// TIA Portal V17 export
// export: Created 2025-03-05T08:00:39.2851451Z, ExportSetting WithDefaults, DisplayName Totally Integrated Automation Portal, DisplayVersion V17 Update 8, DisplayName TIA Portal Openness, DisplayVersion V17 Update 8, DisplayName TIA Portal Version Control Interface, DisplayVersion V17, DisplayName SINAMICS Startdrive Advanced, DisplayVersion V17 SP2, DisplayName SINAMICS Startdrive G110M, G120, G120C, G120D, G120P, G115D, DisplayVersion V17 SP2, DisplayName SINAMICS Startdrive G130, G150, S120, S150, SINAMICS MV, S210, DisplayVersion V17 SP2, DisplayName STEP 7 Professional, DisplayVersion V17 Update 8, DisplayName SINUMERIK ONE STEP 7 Toolbox, DisplayVersion V17 Update 12, DisplayName SINUMERIK 840D sl STEP 7 Toolbox, DisplayVersion V17 Update 12, DisplayName STEP 7 Safety, DisplayVersion V17 Update 6, DisplayName WinCC Advanced, DisplayVersion V17 Update 8
FUNCTION "FC1281_UNIT_02_PART_CHECK_STATION" : Void   // FC1281, LAD
{ S7_Optimized_Access := 'TRUE' }
VERSION : 0.1
// stored: AutoNumber false, IsIECCheckEnabled false, SetENOAutomatically false, UDAEnableTagReadback false
   VAR CONSTANT
      FC_NUMBER : Int := 1281;
   END_VAR
   VAR_TEMP   // added for the SCL form of the ladder/FBD networks
      _w1 : Bool;
      _w2 : Bool;
   END_VAR
BEGIN

REGION Network 1: GENERAL CONDITIONS
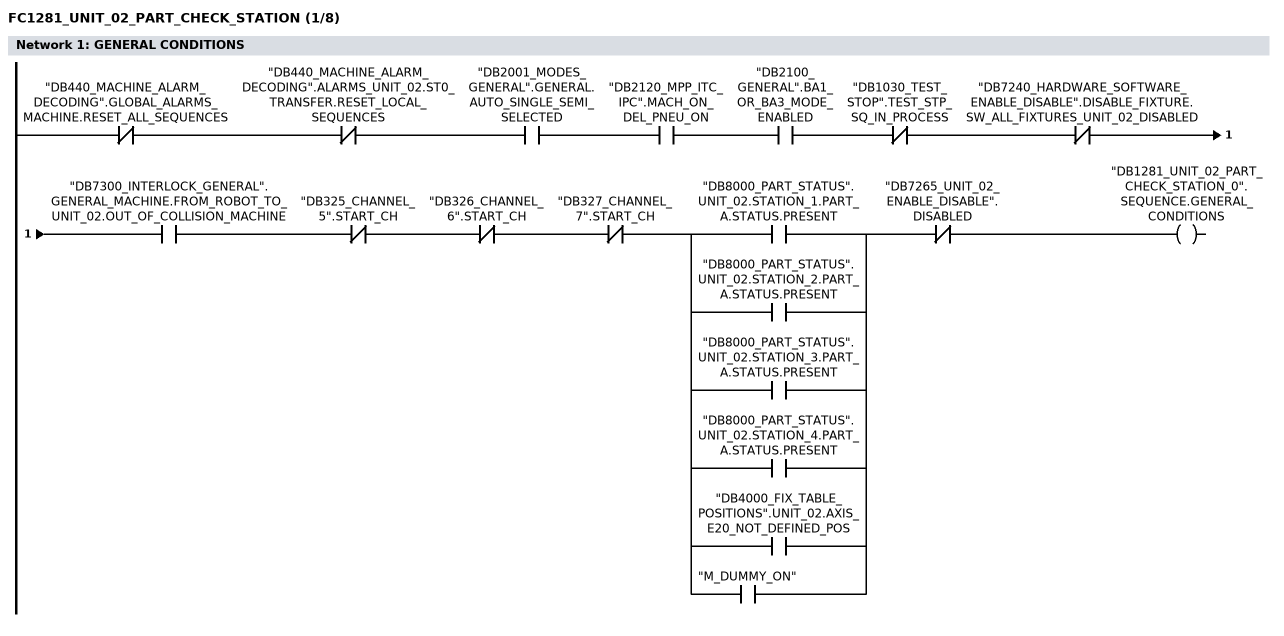
   RUNG wire#powerrail
      I_Contact( "DB440_MACHINE_ALARM_DECODING".GLOBAL_ALARMS_MACHINE.RESET_ALL_SEQUENCES )
      I_Contact( "DB440_MACHINE_ALARM_DECODING".ALARMS_UNIT_02.ST0_TRANSFER.RESET_LOCAL_SEQUENCES )
      Contact( "DB2001_MODES_GENERAL".GENERAL.AUTO_SINGLE_SEMI_SELECTED )
      Contact( "DB2120_MPP_ITC_IPC".MACH_ON_DEL_PNEU_ON )
      Contact( "DB2100_GENERAL".BA1_OR_BA3_MODE_ENABLED )
      I_Contact( "DB1030_TEST_STOP".TEST_STP_SQ_IN_PROCESS )
      I_Contact( "DB7240_HARDWARE_SOFTWARE_ENABLE_DISABLE".DISABLE_FIXTURE.SW_ALL_FIXTURES_UNIT_02_DISABLED )
      Contact( "DB7300_INTERLOCK_GENERAL".GENERAL_MACHINE.FROM_ROBOT_TO_UNIT_02.OUT_OF_COLLISION_MACHINE )
      I_Contact( "DB325_CHANNEL_5".START_CH )
      I_Contact( "DB326_CHANNEL_6".START_CH )
      I_Contact( "DB327_CHANNEL_7".START_CH )
      wire#w1
      Contact( "DB8000_PART_STATUS".UNIT_02.STATION_1.PART_A.STATUS.PRESENT )
      wire#w2
      I_Contact( "DB7265_UNIT_02_ENABLE_DISABLE".DISABLED )
      Coil( "DB1281_UNIT_02_PART_CHECK_STATION_0".SEQUENCE.GENERAL_CONDITIONS )
   END_RUNG
   RUNG wire#w1
      Contact( "DB8000_PART_STATUS".UNIT_02.STATION_2.PART_A.STATUS.PRESENT )
   END_RUNG wire#w2
   RUNG wire#w1
      Contact( "DB8000_PART_STATUS".UNIT_02.STATION_3.PART_A.STATUS.PRESENT )
   END_RUNG wire#w2
   RUNG wire#w1
      Contact( "DB8000_PART_STATUS".UNIT_02.STATION_4.PART_A.STATUS.PRESENT )
   END_RUNG wire#w2
   RUNG wire#w1
      Contact( "DB4000_FIX_TABLE_POSITIONS".UNIT_02.AXIS_E20_NOT_DEFINED_POS )
   END_RUNG wire#w2
   RUNG wire#w1
      Contact( "M_DUMMY_ON" )
   END_RUNG wire#w2
   // the same network as SCL:
   "DB1281_UNIT_02_PART_CHECK_STATION_0".SEQUENCE.GENERAL_CONDITIONS := NOT "DB440_MACHINE_ALARM_DECODING".GLOBAL_ALARMS_MACHINE.RESET_ALL_SEQUENCES AND NOT "DB440_MACHINE_ALARM_DECODING".ALARMS_UNIT_02.ST0_TRANSFER.RESET_LOCAL_SEQUENCES AND "DB2001_MODES_GENERAL".GENERAL.AUTO_SINGLE_SEMI_SELECTED AND "DB2120_MPP_ITC_IPC".MACH_ON_DEL_PNEU_ON AND "DB2100_GENERAL".BA1_OR_BA3_MODE_ENABLED AND NOT "DB1030_TEST_STOP".TEST_STP_SQ_IN_PROCESS AND NOT "DB7240_HARDWARE_SOFTWARE_ENABLE_DISABLE".DISABLE_FIXTURE.SW_ALL_FIXTURES_UNIT_02_DISABLED AND "DB7300_INTERLOCK_GENERAL".GENERAL_MACHINE.FROM_ROBOT_TO_UNIT_02.OUT_OF_COLLISION_MACHINE AND NOT "DB325_CHANNEL_5".START_CH AND NOT "DB326_CHANNEL_6".START_CH AND NOT "DB327_CHANNEL_7".START_CH AND ("DB8000_PART_STATUS".UNIT_02.STATION_1.PART_A.STATUS.PRESENT OR "DB8000_PART_STATUS".UNIT_02.STATION_2.PART_A.STATUS.PRESENT OR "DB8000_PART_STATUS".UNIT_02.STATION_3.PART_A.STATUS.PRESENT OR "DB8000_PART_STATUS".UNIT_02.STATION_4.PART_A.STATUS.PRESENT OR "DB4000_FIX_TABLE_POSITIONS".UNIT_02.AXIS_E20_NOT_DEFINED_POS OR "M_DUMMY_ON") AND NOT "DB7265_UNIT_02_ENABLE_DISABLE".DISABLED;
END_REGION

REGION Network 2: OPERATOR HELP
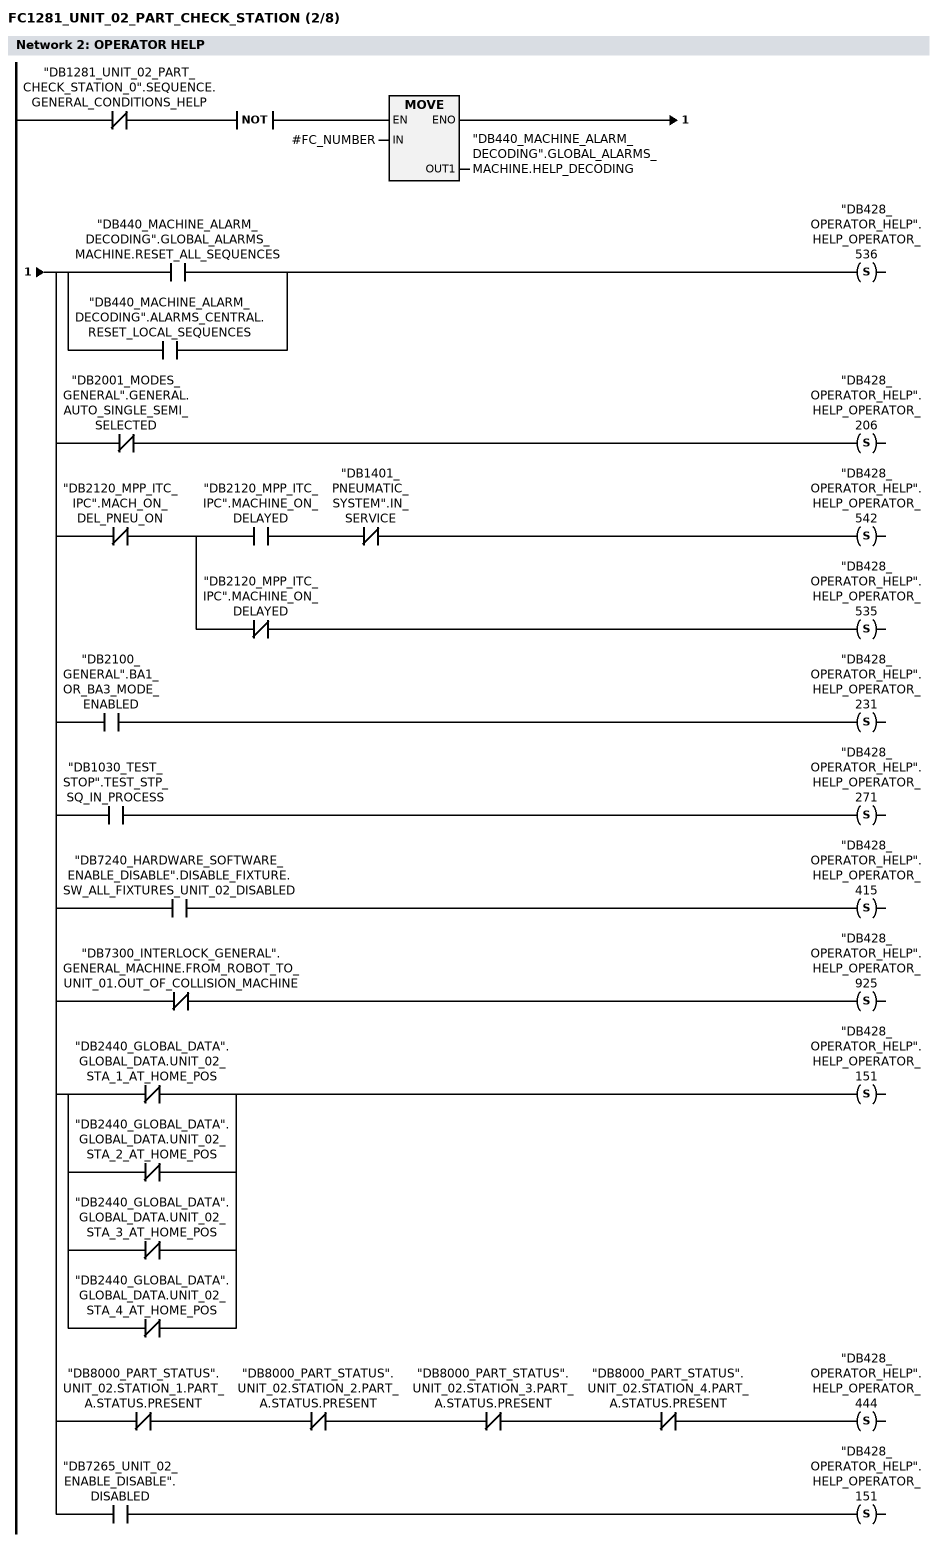
   RUNG wire#powerrail
      I_Contact( "DB1281_UNIT_02_PART_CHECK_STATION_0".SEQUENCE.GENERAL_CONDITIONS_HELP )
      Not()
      { S7_GenerateENO := "TRUE" } Move(in := #FC_NUMBER, out1 => "DB440_MACHINE_ALARM_DECODING".GLOBAL_ALARMS_MACHINE.HELP_DECODING)
      wire#w1
      Contact( "DB440_MACHINE_ALARM_DECODING".GLOBAL_ALARMS_MACHINE.RESET_ALL_SEQUENCES )
      wire#w2
      S_Coil( "DB428_OPERATOR_HELP".HELP_OPERATOR_536 )
   END_RUNG
   RUNG wire#w1
      Contact( "DB440_MACHINE_ALARM_DECODING".ALARMS_CENTRAL.RESET_LOCAL_SEQUENCES )
   END_RUNG wire#w2
   RUNG wire#w1
      I_Contact( "DB2001_MODES_GENERAL".GENERAL.AUTO_SINGLE_SEMI_SELECTED )
      S_Coil( "DB428_OPERATOR_HELP".HELP_OPERATOR_206 )
   END_RUNG
   RUNG wire#w1
      I_Contact( "DB2120_MPP_ITC_IPC".MACH_ON_DEL_PNEU_ON )
      wire#w3
      Contact( "DB2120_MPP_ITC_IPC".MACHINE_ON_DELAYED )
      I_Contact( "DB1401_PNEUMATIC_SYSTEM".IN_SERVICE )
      S_Coil( "DB428_OPERATOR_HELP".HELP_OPERATOR_542 )
   END_RUNG
   RUNG wire#w3
      I_Contact( "DB2120_MPP_ITC_IPC".MACHINE_ON_DELAYED )
      S_Coil( "DB428_OPERATOR_HELP".HELP_OPERATOR_535 )
   END_RUNG
   RUNG wire#w1
      Contact( "DB2100_GENERAL".BA1_OR_BA3_MODE_ENABLED )
      S_Coil( "DB428_OPERATOR_HELP".HELP_OPERATOR_231 )
   END_RUNG
   RUNG wire#w1
      Contact( "DB1030_TEST_STOP".TEST_STP_SQ_IN_PROCESS )
      S_Coil( "DB428_OPERATOR_HELP".HELP_OPERATOR_271 )
   END_RUNG
   RUNG wire#w1
      Contact( "DB7240_HARDWARE_SOFTWARE_ENABLE_DISABLE".DISABLE_FIXTURE.SW_ALL_FIXTURES_UNIT_02_DISABLED )
      S_Coil( "DB428_OPERATOR_HELP".HELP_OPERATOR_415 )
   END_RUNG
   RUNG wire#w1
      I_Contact( "DB7300_INTERLOCK_GENERAL".GENERAL_MACHINE.FROM_ROBOT_TO_UNIT_01.OUT_OF_COLLISION_MACHINE )
      S_Coil( "DB428_OPERATOR_HELP".HELP_OPERATOR_925 )
   END_RUNG
   RUNG wire#w1
      I_Contact( "DB2440_GLOBAL_DATA".GLOBAL_DATA.UNIT_02_STA_1_AT_HOME_POS )
      wire#w4
      S_Coil( "DB428_OPERATOR_HELP".HELP_OPERATOR_151 )
   END_RUNG
   RUNG wire#w1
      I_Contact( "DB2440_GLOBAL_DATA".GLOBAL_DATA.UNIT_02_STA_2_AT_HOME_POS )
   END_RUNG wire#w4
   RUNG wire#w1
      I_Contact( "DB2440_GLOBAL_DATA".GLOBAL_DATA.UNIT_02_STA_3_AT_HOME_POS )
   END_RUNG wire#w4
   RUNG wire#w1
      I_Contact( "DB2440_GLOBAL_DATA".GLOBAL_DATA.UNIT_02_STA_4_AT_HOME_POS )
   END_RUNG wire#w4
   RUNG wire#w1
      I_Contact( "DB8000_PART_STATUS".UNIT_02.STATION_1.PART_A.STATUS.PRESENT )
      I_Contact( "DB8000_PART_STATUS".UNIT_02.STATION_2.PART_A.STATUS.PRESENT )
      I_Contact( "DB8000_PART_STATUS".UNIT_02.STATION_3.PART_A.STATUS.PRESENT )
      I_Contact( "DB8000_PART_STATUS".UNIT_02.STATION_4.PART_A.STATUS.PRESENT )
      S_Coil( "DB428_OPERATOR_HELP".HELP_OPERATOR_444 )
   END_RUNG
   RUNG wire#w1
      Contact( "DB7265_UNIT_02_ENABLE_DISABLE".DISABLED )
      S_Coil( "DB428_OPERATOR_HELP".HELP_OPERATOR_151 )
   END_RUNG
   // the same network as SCL:
   // ENO of a box is taken as its EN; it also drops when the box reports an error
   #_w1 := NOT (NOT "DB1281_UNIT_02_PART_CHECK_STATION_0".SEQUENCE.GENERAL_CONDITIONS_HELP);
   IF #_w1 THEN "DB440_MACHINE_ALARM_DECODING".GLOBAL_ALARMS_MACHINE.HELP_DECODING := #FC_NUMBER; END_IF;
   IF #_w1 AND ("DB440_MACHINE_ALARM_DECODING".GLOBAL_ALARMS_MACHINE.RESET_ALL_SEQUENCES OR "DB440_MACHINE_ALARM_DECODING".ALARMS_CENTRAL.RESET_LOCAL_SEQUENCES) THEN
       "DB428_OPERATOR_HELP".HELP_OPERATOR_536 := TRUE;
   END_IF;
   IF #_w1 AND NOT "DB2001_MODES_GENERAL".GENERAL.AUTO_SINGLE_SEMI_SELECTED THEN
       "DB428_OPERATOR_HELP".HELP_OPERATOR_206 := TRUE;
   END_IF;
   #_w2 := #_w1 AND NOT "DB2120_MPP_ITC_IPC".MACH_ON_DEL_PNEU_ON;
   IF #_w2 AND "DB2120_MPP_ITC_IPC".MACHINE_ON_DELAYED AND NOT "DB1401_PNEUMATIC_SYSTEM".IN_SERVICE THEN
       "DB428_OPERATOR_HELP".HELP_OPERATOR_542 := TRUE;
   END_IF;
   IF #_w2 AND NOT "DB2120_MPP_ITC_IPC".MACHINE_ON_DELAYED THEN
       "DB428_OPERATOR_HELP".HELP_OPERATOR_535 := TRUE;
   END_IF;
   IF #_w1 AND "DB2100_GENERAL".BA1_OR_BA3_MODE_ENABLED THEN
       "DB428_OPERATOR_HELP".HELP_OPERATOR_231 := TRUE;
   END_IF;
   IF #_w1 AND "DB1030_TEST_STOP".TEST_STP_SQ_IN_PROCESS THEN
       "DB428_OPERATOR_HELP".HELP_OPERATOR_271 := TRUE;
   END_IF;
   IF #_w1 AND "DB7240_HARDWARE_SOFTWARE_ENABLE_DISABLE".DISABLE_FIXTURE.SW_ALL_FIXTURES_UNIT_02_DISABLED THEN
       "DB428_OPERATOR_HELP".HELP_OPERATOR_415 := TRUE;
   END_IF;
   IF #_w1 AND NOT "DB7300_INTERLOCK_GENERAL".GENERAL_MACHINE.FROM_ROBOT_TO_UNIT_01.OUT_OF_COLLISION_MACHINE THEN
       "DB428_OPERATOR_HELP".HELP_OPERATOR_925 := TRUE;
   END_IF;
   IF #_w1 AND (NOT "DB2440_GLOBAL_DATA".GLOBAL_DATA.UNIT_02_STA_1_AT_HOME_POS OR NOT "DB2440_GLOBAL_DATA".GLOBAL_DATA.UNIT_02_STA_2_AT_HOME_POS OR NOT "DB2440_GLOBAL_DATA".GLOBAL_DATA.UNIT_02_STA_3_AT_HOME_POS OR NOT "DB2440_GLOBAL_DATA".GLOBAL_DATA.UNIT_02_STA_4_AT_HOME_POS) THEN
       "DB428_OPERATOR_HELP".HELP_OPERATOR_151 := TRUE;
   END_IF;
   IF #_w1 AND NOT "DB8000_PART_STATUS".UNIT_02.STATION_1.PART_A.STATUS.PRESENT AND NOT "DB8000_PART_STATUS".UNIT_02.STATION_2.PART_A.STATUS.PRESENT AND NOT "DB8000_PART_STATUS".UNIT_02.STATION_3.PART_A.STATUS.PRESENT AND NOT "DB8000_PART_STATUS".UNIT_02.STATION_4.PART_A.STATUS.PRESENT THEN
       "DB428_OPERATOR_HELP".HELP_OPERATOR_444 := TRUE;
   END_IF;
   IF #_w1 AND "DB7265_UNIT_02_ENABLE_DISABLE".DISABLED THEN
       "DB428_OPERATOR_HELP".HELP_OPERATOR_151 := TRUE;
   END_IF;
END_REGION

REGION Network 3: INITIAL CONDITIONS
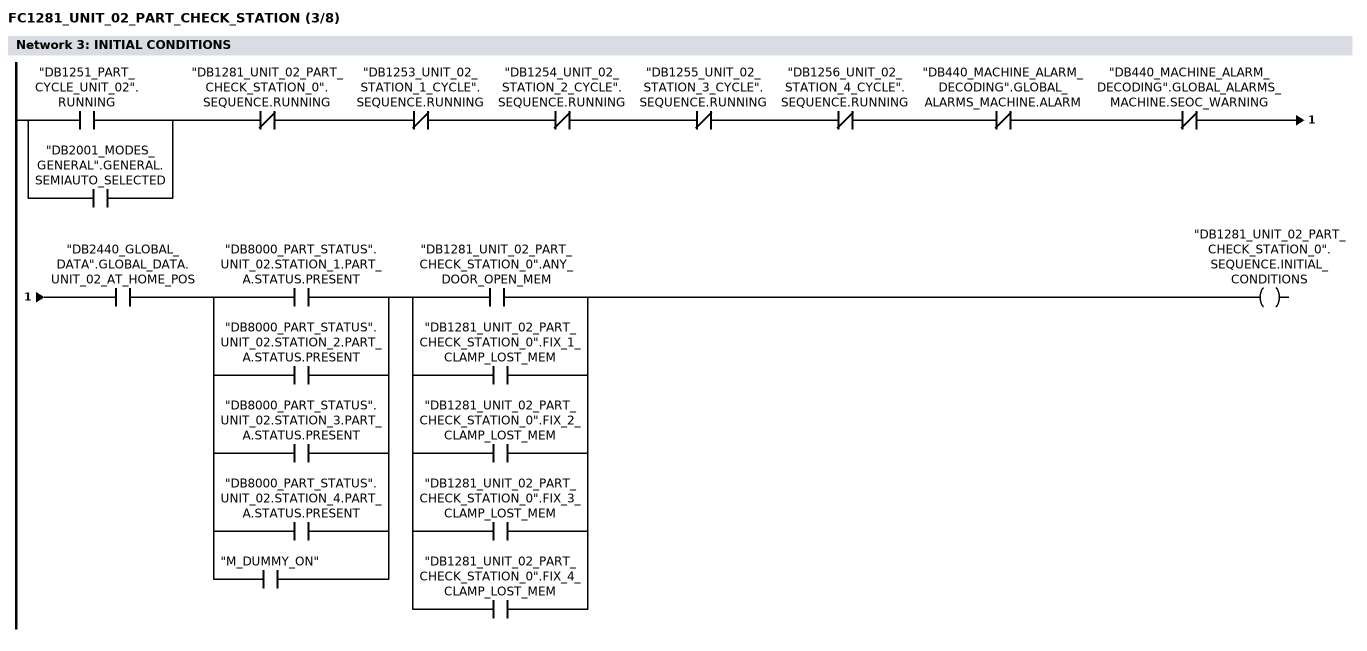
   RUNG wire#powerrail
      Contact( "DB1251_PART_CYCLE_UNIT_02".RUNNING )
      wire#w1
      I_Contact( "DB1281_UNIT_02_PART_CHECK_STATION_0".SEQUENCE.RUNNING )
      I_Contact( "DB1253_UNIT_02_STATION_1_CYCLE".SEQUENCE.RUNNING )
      I_Contact( "DB1254_UNIT_02_STATION_2_CYCLE".SEQUENCE.RUNNING )
      I_Contact( "DB1255_UNIT_02_STATION_3_CYCLE".SEQUENCE.RUNNING )
      I_Contact( "DB1256_UNIT_02_STATION_4_CYCLE".SEQUENCE.RUNNING )
      I_Contact( "DB440_MACHINE_ALARM_DECODING".GLOBAL_ALARMS_MACHINE.ALARM )
      I_Contact( "DB440_MACHINE_ALARM_DECODING".GLOBAL_ALARMS_MACHINE.SEOC_WARNING )
      Contact( "DB2440_GLOBAL_DATA".GLOBAL_DATA.UNIT_02_AT_HOME_POS )
      wire#w2
      Contact( "DB8000_PART_STATUS".UNIT_02.STATION_1.PART_A.STATUS.PRESENT )
      wire#w3
      Contact( "DB1281_UNIT_02_PART_CHECK_STATION_0".ANY_DOOR_OPEN_MEM )
      wire#w4
      Coil( "DB1281_UNIT_02_PART_CHECK_STATION_0".SEQUENCE.INITIAL_CONDITIONS )
   END_RUNG
   RUNG wire#powerrail
      Contact( "DB2001_MODES_GENERAL".GENERAL.SEMIAUTO_SELECTED )
   END_RUNG wire#w1
   RUNG wire#w2
      Contact( "DB8000_PART_STATUS".UNIT_02.STATION_2.PART_A.STATUS.PRESENT )
   END_RUNG wire#w3
   RUNG wire#w2
      Contact( "DB8000_PART_STATUS".UNIT_02.STATION_3.PART_A.STATUS.PRESENT )
   END_RUNG wire#w3
   RUNG wire#w2
      Contact( "DB8000_PART_STATUS".UNIT_02.STATION_4.PART_A.STATUS.PRESENT )
   END_RUNG wire#w3
   RUNG wire#w2
      Contact( "M_DUMMY_ON" )
   END_RUNG wire#w3
   RUNG wire#w3
      Contact( "DB1281_UNIT_02_PART_CHECK_STATION_0".FIX_1_CLAMP_LOST_MEM )
   END_RUNG wire#w4
   RUNG wire#w3
      Contact( "DB1281_UNIT_02_PART_CHECK_STATION_0".FIX_2_CLAMP_LOST_MEM )
   END_RUNG wire#w4
   RUNG wire#w3
      Contact( "DB1281_UNIT_02_PART_CHECK_STATION_0".FIX_3_CLAMP_LOST_MEM )
   END_RUNG wire#w4
   RUNG wire#w3
      Contact( "DB1281_UNIT_02_PART_CHECK_STATION_0".FIX_4_CLAMP_LOST_MEM )
   END_RUNG wire#w4
   // the same network as SCL:
   "DB1281_UNIT_02_PART_CHECK_STATION_0".SEQUENCE.INITIAL_CONDITIONS := ("DB1251_PART_CYCLE_UNIT_02".RUNNING OR "DB2001_MODES_GENERAL".GENERAL.SEMIAUTO_SELECTED) AND NOT "DB1281_UNIT_02_PART_CHECK_STATION_0".SEQUENCE.RUNNING AND NOT "DB1253_UNIT_02_STATION_1_CYCLE".SEQUENCE.RUNNING AND NOT "DB1254_UNIT_02_STATION_2_CYCLE".SEQUENCE.RUNNING AND NOT "DB1255_UNIT_02_STATION_3_CYCLE".SEQUENCE.RUNNING AND NOT "DB1256_UNIT_02_STATION_4_CYCLE".SEQUENCE.RUNNING AND NOT "DB440_MACHINE_ALARM_DECODING".GLOBAL_ALARMS_MACHINE.ALARM AND NOT "DB440_MACHINE_ALARM_DECODING".GLOBAL_ALARMS_MACHINE.SEOC_WARNING AND "DB2440_GLOBAL_DATA".GLOBAL_DATA.UNIT_02_AT_HOME_POS AND ("DB8000_PART_STATUS".UNIT_02.STATION_1.PART_A.STATUS.PRESENT OR "DB8000_PART_STATUS".UNIT_02.STATION_2.PART_A.STATUS.PRESENT OR "DB8000_PART_STATUS".UNIT_02.STATION_3.PART_A.STATUS.PRESENT OR "DB8000_PART_STATUS".UNIT_02.STATION_4.PART_A.STATUS.PRESENT OR "M_DUMMY_ON") AND ("DB1281_UNIT_02_PART_CHECK_STATION_0".ANY_DOOR_OPEN_MEM OR "DB1281_UNIT_02_PART_CHECK_STATION_0".FIX_1_CLAMP_LOST_MEM OR "DB1281_UNIT_02_PART_CHECK_STATION_0".FIX_2_CLAMP_LOST_MEM OR "DB1281_UNIT_02_PART_CHECK_STATION_0".FIX_3_CLAMP_LOST_MEM OR "DB1281_UNIT_02_PART_CHECK_STATION_0".FIX_4_CLAMP_LOST_MEM);
END_REGION

REGION Network 4: OPERATOR HELP
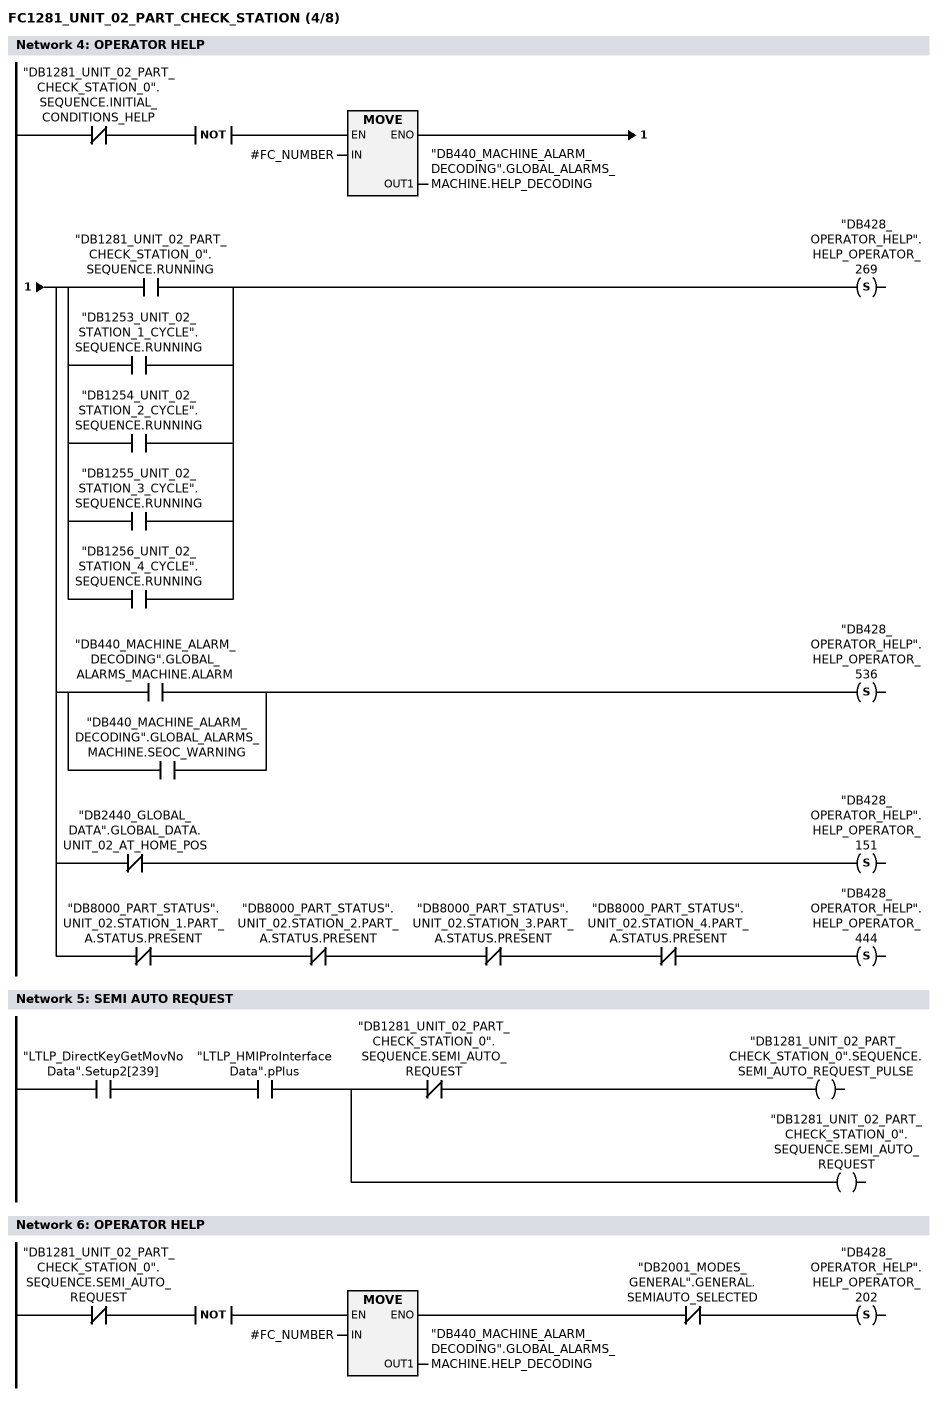
   RUNG wire#powerrail
      I_Contact( "DB1281_UNIT_02_PART_CHECK_STATION_0".SEQUENCE.INITIAL_CONDITIONS_HELP )
      Not()
      { S7_GenerateENO := "TRUE" } Move(in := #FC_NUMBER, out1 => "DB440_MACHINE_ALARM_DECODING".GLOBAL_ALARMS_MACHINE.HELP_DECODING)
      wire#w1
      Contact( "DB1281_UNIT_02_PART_CHECK_STATION_0".SEQUENCE.RUNNING )
      wire#w2
      S_Coil( "DB428_OPERATOR_HELP".HELP_OPERATOR_269 )
   END_RUNG
   RUNG wire#w1
      Contact( "DB1253_UNIT_02_STATION_1_CYCLE".SEQUENCE.RUNNING )
   END_RUNG wire#w2
   RUNG wire#w1
      Contact( "DB1254_UNIT_02_STATION_2_CYCLE".SEQUENCE.RUNNING )
   END_RUNG wire#w2
   RUNG wire#w1
      Contact( "DB1255_UNIT_02_STATION_3_CYCLE".SEQUENCE.RUNNING )
   END_RUNG wire#w2
   RUNG wire#w1
      Contact( "DB1256_UNIT_02_STATION_4_CYCLE".SEQUENCE.RUNNING )
   END_RUNG wire#w2
   RUNG wire#w1
      Contact( "DB440_MACHINE_ALARM_DECODING".GLOBAL_ALARMS_MACHINE.ALARM )
      wire#w3
      S_Coil( "DB428_OPERATOR_HELP".HELP_OPERATOR_536 )
   END_RUNG
   RUNG wire#w1
      Contact( "DB440_MACHINE_ALARM_DECODING".GLOBAL_ALARMS_MACHINE.SEOC_WARNING )
   END_RUNG wire#w3
   RUNG wire#w1
      I_Contact( "DB2440_GLOBAL_DATA".GLOBAL_DATA.UNIT_02_AT_HOME_POS )
      S_Coil( "DB428_OPERATOR_HELP".HELP_OPERATOR_151 )
   END_RUNG
   RUNG wire#w1
      I_Contact( "DB8000_PART_STATUS".UNIT_02.STATION_1.PART_A.STATUS.PRESENT )
      I_Contact( "DB8000_PART_STATUS".UNIT_02.STATION_2.PART_A.STATUS.PRESENT )
      I_Contact( "DB8000_PART_STATUS".UNIT_02.STATION_3.PART_A.STATUS.PRESENT )
      I_Contact( "DB8000_PART_STATUS".UNIT_02.STATION_4.PART_A.STATUS.PRESENT )
      S_Coil( "DB428_OPERATOR_HELP".HELP_OPERATOR_444 )
   END_RUNG
   // the same network as SCL:
   // ENO of a box is taken as its EN; it also drops when the box reports an error
   #_w1 := NOT (NOT "DB1281_UNIT_02_PART_CHECK_STATION_0".SEQUENCE.INITIAL_CONDITIONS_HELP);
   IF #_w1 THEN "DB440_MACHINE_ALARM_DECODING".GLOBAL_ALARMS_MACHINE.HELP_DECODING := #FC_NUMBER; END_IF;
   IF #_w1 AND ("DB1281_UNIT_02_PART_CHECK_STATION_0".SEQUENCE.RUNNING OR "DB1253_UNIT_02_STATION_1_CYCLE".SEQUENCE.RUNNING OR "DB1254_UNIT_02_STATION_2_CYCLE".SEQUENCE.RUNNING OR "DB1255_UNIT_02_STATION_3_CYCLE".SEQUENCE.RUNNING OR "DB1256_UNIT_02_STATION_4_CYCLE".SEQUENCE.RUNNING) THEN
       "DB428_OPERATOR_HELP".HELP_OPERATOR_269 := TRUE;
   END_IF;
   IF #_w1 AND ("DB440_MACHINE_ALARM_DECODING".GLOBAL_ALARMS_MACHINE.ALARM OR "DB440_MACHINE_ALARM_DECODING".GLOBAL_ALARMS_MACHINE.SEOC_WARNING) THEN
       "DB428_OPERATOR_HELP".HELP_OPERATOR_536 := TRUE;
   END_IF;
   IF #_w1 AND NOT "DB2440_GLOBAL_DATA".GLOBAL_DATA.UNIT_02_AT_HOME_POS THEN
       "DB428_OPERATOR_HELP".HELP_OPERATOR_151 := TRUE;
   END_IF;
   IF #_w1 AND NOT "DB8000_PART_STATUS".UNIT_02.STATION_1.PART_A.STATUS.PRESENT AND NOT "DB8000_PART_STATUS".UNIT_02.STATION_2.PART_A.STATUS.PRESENT AND NOT "DB8000_PART_STATUS".UNIT_02.STATION_3.PART_A.STATUS.PRESENT AND NOT "DB8000_PART_STATUS".UNIT_02.STATION_4.PART_A.STATUS.PRESENT THEN
       "DB428_OPERATOR_HELP".HELP_OPERATOR_444 := TRUE;
   END_IF;
END_REGION

REGION Network 5: SEMI AUTO REQUEST
   RUNG wire#powerrail
      Contact( "LTLP_DirectKeyGetMovNoData".Setup2[239] )
      Contact( "LTLP_HMIProInterfaceData".pPlus )
      wire#w1
      I_Contact( "DB1281_UNIT_02_PART_CHECK_STATION_0".SEQUENCE.SEMI_AUTO_REQUEST )
      Coil( "DB1281_UNIT_02_PART_CHECK_STATION_0".SEQUENCE.SEMI_AUTO_REQUEST_PULSE )
   END_RUNG
   RUNG wire#w1
      Coil( "DB1281_UNIT_02_PART_CHECK_STATION_0".SEQUENCE.SEMI_AUTO_REQUEST )
   END_RUNG
   // the same network as SCL:
   #_w1 := "LTLP_DirectKeyGetMovNoData".Setup2[239] AND "LTLP_HMIProInterfaceData".pPlus;
   "DB1281_UNIT_02_PART_CHECK_STATION_0".SEQUENCE.SEMI_AUTO_REQUEST_PULSE := #_w1 AND NOT "DB1281_UNIT_02_PART_CHECK_STATION_0".SEQUENCE.SEMI_AUTO_REQUEST;
   "DB1281_UNIT_02_PART_CHECK_STATION_0".SEQUENCE.SEMI_AUTO_REQUEST := #_w1;
END_REGION

REGION Network 6: OPERATOR HELP
   RUNG wire#powerrail
      I_Contact( "DB1281_UNIT_02_PART_CHECK_STATION_0".SEQUENCE.SEMI_AUTO_REQUEST )
      Not()
      { S7_GenerateENO := "TRUE" } Move(in := #FC_NUMBER, out1 => "DB440_MACHINE_ALARM_DECODING".GLOBAL_ALARMS_MACHINE.HELP_DECODING)
      I_Contact( "DB2001_MODES_GENERAL".GENERAL.SEMIAUTO_SELECTED )
      S_Coil( "DB428_OPERATOR_HELP".HELP_OPERATOR_202 )
   END_RUNG
   // the same network as SCL:
   // ENO of a box is taken as its EN; it also drops when the box reports an error
   #_w1 := NOT (NOT "DB1281_UNIT_02_PART_CHECK_STATION_0".SEQUENCE.SEMI_AUTO_REQUEST);
   IF #_w1 THEN "DB440_MACHINE_ALARM_DECODING".GLOBAL_ALARMS_MACHINE.HELP_DECODING := #FC_NUMBER; END_IF;
   IF #_w1 AND NOT "DB2001_MODES_GENERAL".GENERAL.SEMIAUTO_SELECTED THEN
       "DB428_OPERATOR_HELP".HELP_OPERATOR_202 := TRUE;
   END_IF;
END_REGION

REGION Network 7: ANY DOOR OPEN MEMORY
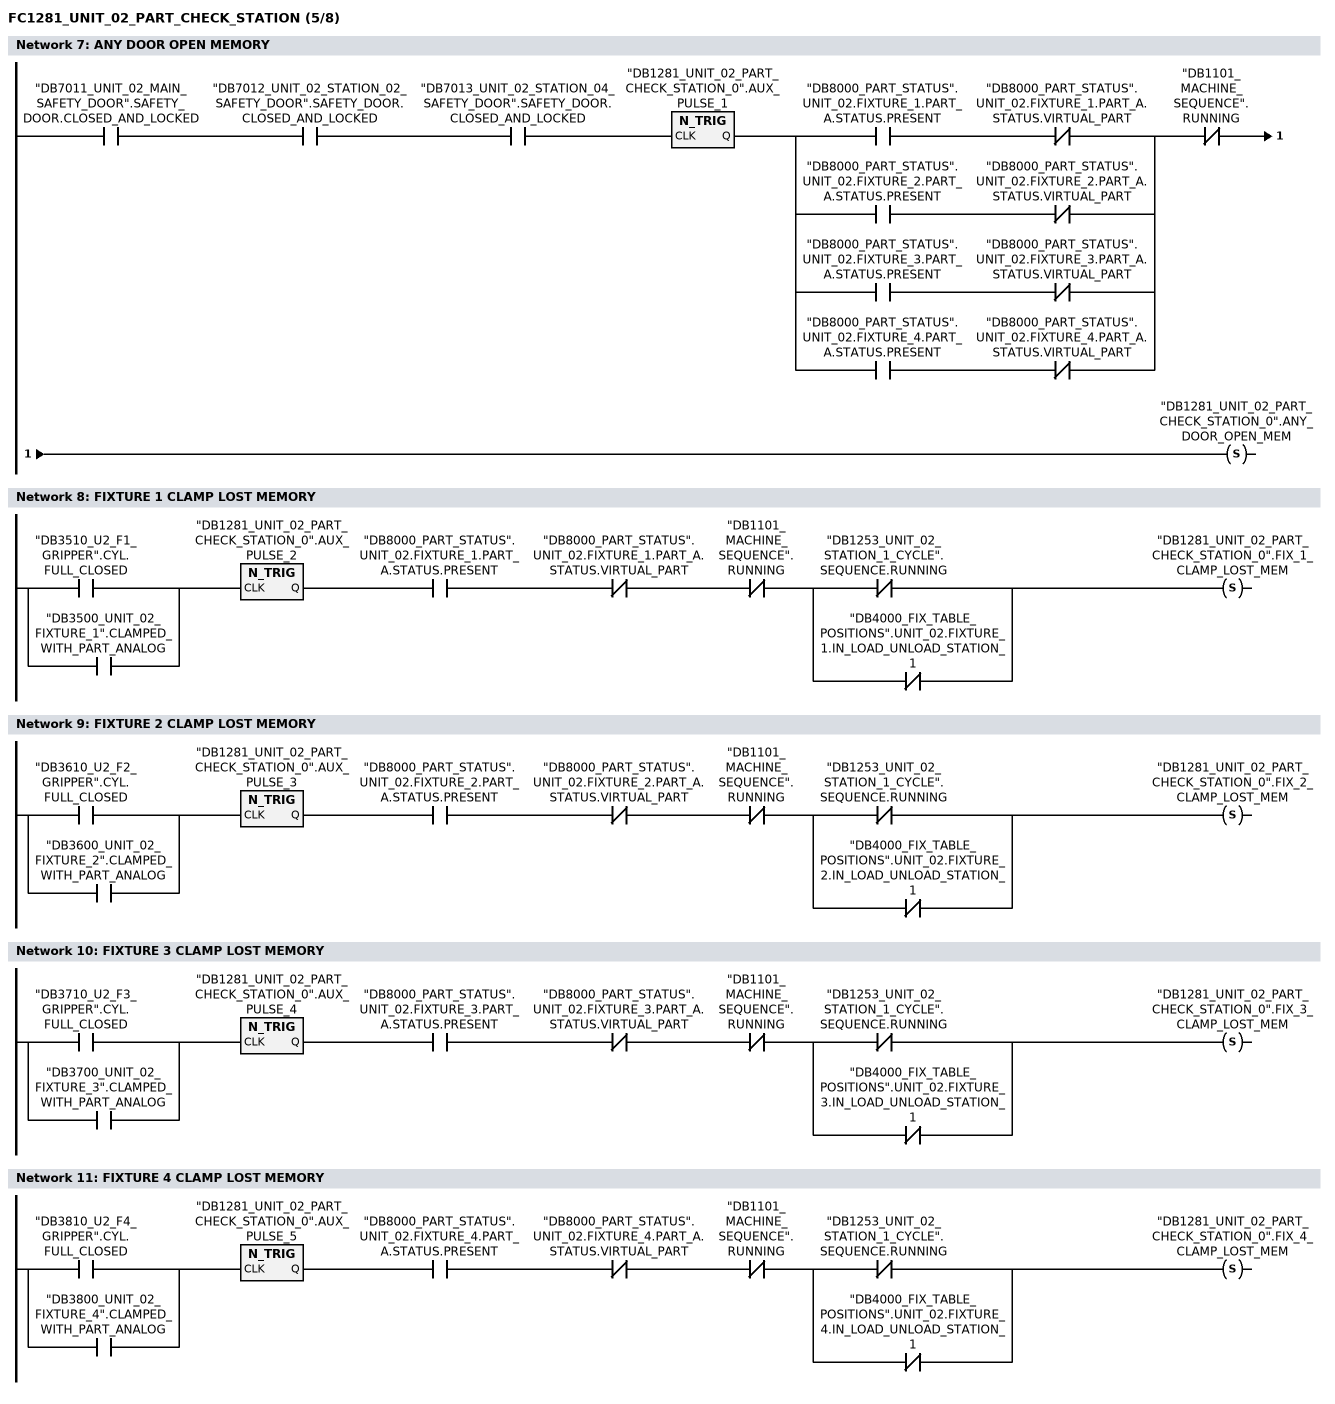
   RUNG wire#powerrail
      Contact( "DB7011_UNIT_02_MAIN_SAFETY_DOOR".SAFETY_DOOR.CLOSED_AND_LOCKED )
      Contact( "DB7012_UNIT_02_STATION_02_SAFETY_DOOR".SAFETY_DOOR.CLOSED_AND_LOCKED )
      Contact( "DB7013_UNIT_02_STATION_04_SAFETY_DOOR".SAFETY_DOOR.CLOSED_AND_LOCKED )
      N_Trig( "DB1281_UNIT_02_PART_CHECK_STATION_0".AUX_PULSE_1 )
      wire#w1
      Contact( "DB8000_PART_STATUS".UNIT_02.FIXTURE_1.PART_A.STATUS.PRESENT )
      I_Contact( "DB8000_PART_STATUS".UNIT_02.FIXTURE_1.PART_A.STATUS.VIRTUAL_PART )
      wire#w2
      I_Contact( "DB1101_MACHINE_SEQUENCE".RUNNING )
      S_Coil( "DB1281_UNIT_02_PART_CHECK_STATION_0".ANY_DOOR_OPEN_MEM )
   END_RUNG
   RUNG wire#w1
      Contact( "DB8000_PART_STATUS".UNIT_02.FIXTURE_2.PART_A.STATUS.PRESENT )
      I_Contact( "DB8000_PART_STATUS".UNIT_02.FIXTURE_2.PART_A.STATUS.VIRTUAL_PART )
   END_RUNG wire#w2
   RUNG wire#w1
      Contact( "DB8000_PART_STATUS".UNIT_02.FIXTURE_3.PART_A.STATUS.PRESENT )
      I_Contact( "DB8000_PART_STATUS".UNIT_02.FIXTURE_3.PART_A.STATUS.VIRTUAL_PART )
   END_RUNG wire#w2
   RUNG wire#w1
      Contact( "DB8000_PART_STATUS".UNIT_02.FIXTURE_4.PART_A.STATUS.PRESENT )
      I_Contact( "DB8000_PART_STATUS".UNIT_02.FIXTURE_4.PART_A.STATUS.VIRTUAL_PART )
   END_RUNG wire#w2
   // the same network as SCL:
   #_w1 := "DB7011_UNIT_02_MAIN_SAFETY_DOOR".SAFETY_DOOR.CLOSED_AND_LOCKED AND "DB7012_UNIT_02_STATION_02_SAFETY_DOOR".SAFETY_DOOR.CLOSED_AND_LOCKED AND "DB7013_UNIT_02_STATION_04_SAFETY_DOOR".SAFETY_DOOR.CLOSED_AND_LOCKED;
   #_w2 := NOT #_w1 AND "DB1281_UNIT_02_PART_CHECK_STATION_0".AUX_PULSE_1;   // falling edge
   "DB1281_UNIT_02_PART_CHECK_STATION_0".AUX_PULSE_1 := #_w1;
   IF #_w2 AND (("DB8000_PART_STATUS".UNIT_02.FIXTURE_1.PART_A.STATUS.PRESENT AND NOT "DB8000_PART_STATUS".UNIT_02.FIXTURE_1.PART_A.STATUS.VIRTUAL_PART) OR ("DB8000_PART_STATUS".UNIT_02.FIXTURE_2.PART_A.STATUS.PRESENT AND NOT "DB8000_PART_STATUS".UNIT_02.FIXTURE_2.PART_A.STATUS.VIRTUAL_PART) OR ("DB8000_PART_STATUS".UNIT_02.FIXTURE_3.PART_A.STATUS.PRESENT AND NOT "DB8000_PART_STATUS".UNIT_02.FIXTURE_3.PART_A.STATUS.VIRTUAL_PART) OR ("DB8000_PART_STATUS".UNIT_02.FIXTURE_4.PART_A.STATUS.PRESENT AND NOT "DB8000_PART_STATUS".UNIT_02.FIXTURE_4.PART_A.STATUS.VIRTUAL_PART)) AND NOT "DB1101_MACHINE_SEQUENCE".RUNNING THEN
       "DB1281_UNIT_02_PART_CHECK_STATION_0".ANY_DOOR_OPEN_MEM := TRUE;
   END_IF;
END_REGION

REGION Network 8: FIXTURE 1 CLAMP LOST MEMORY
   RUNG wire#powerrail
      Contact( "DB3510_U2_F1_GRIPPER".CYL.FULL_CLOSED )
      wire#w1
      N_Trig( "DB1281_UNIT_02_PART_CHECK_STATION_0".AUX_PULSE_2 )
      Contact( "DB8000_PART_STATUS".UNIT_02.FIXTURE_1.PART_A.STATUS.PRESENT )
      I_Contact( "DB8000_PART_STATUS".UNIT_02.FIXTURE_1.PART_A.STATUS.VIRTUAL_PART )
      I_Contact( "DB1101_MACHINE_SEQUENCE".RUNNING )
      wire#w2
      I_Contact( "DB1253_UNIT_02_STATION_1_CYCLE".SEQUENCE.RUNNING )
      wire#w3
      S_Coil( "DB1281_UNIT_02_PART_CHECK_STATION_0".FIX_1_CLAMP_LOST_MEM )
   END_RUNG
   RUNG wire#powerrail
      Contact( "DB3500_UNIT_02_FIXTURE_1".CLAMPED_WITH_PART_ANALOG )
   END_RUNG wire#w1
   RUNG wire#w2
      I_Contact( "DB4000_FIX_TABLE_POSITIONS".UNIT_02.FIXTURE_1.IN_LOAD_UNLOAD_STATION_1 )
   END_RUNG wire#w3
   // the same network as SCL:
   #_w1 := "DB3510_U2_F1_GRIPPER".CYL.FULL_CLOSED OR "DB3500_UNIT_02_FIXTURE_1".CLAMPED_WITH_PART_ANALOG;
   #_w2 := NOT #_w1 AND "DB1281_UNIT_02_PART_CHECK_STATION_0".AUX_PULSE_2;   // falling edge
   "DB1281_UNIT_02_PART_CHECK_STATION_0".AUX_PULSE_2 := #_w1;
   IF #_w2 AND "DB8000_PART_STATUS".UNIT_02.FIXTURE_1.PART_A.STATUS.PRESENT AND NOT "DB8000_PART_STATUS".UNIT_02.FIXTURE_1.PART_A.STATUS.VIRTUAL_PART AND NOT "DB1101_MACHINE_SEQUENCE".RUNNING AND (NOT "DB1253_UNIT_02_STATION_1_CYCLE".SEQUENCE.RUNNING OR NOT "DB4000_FIX_TABLE_POSITIONS".UNIT_02.FIXTURE_1.IN_LOAD_UNLOAD_STATION_1) THEN
       "DB1281_UNIT_02_PART_CHECK_STATION_0".FIX_1_CLAMP_LOST_MEM := TRUE;
   END_IF;
END_REGION

REGION Network 9: FIXTURE 2 CLAMP LOST MEMORY
   RUNG wire#powerrail
      Contact( "DB3610_U2_F2_GRIPPER".CYL.FULL_CLOSED )
      wire#w1
      N_Trig( "DB1281_UNIT_02_PART_CHECK_STATION_0".AUX_PULSE_3 )
      Contact( "DB8000_PART_STATUS".UNIT_02.FIXTURE_2.PART_A.STATUS.PRESENT )
      I_Contact( "DB8000_PART_STATUS".UNIT_02.FIXTURE_2.PART_A.STATUS.VIRTUAL_PART )
      I_Contact( "DB1101_MACHINE_SEQUENCE".RUNNING )
      wire#w2
      I_Contact( "DB1253_UNIT_02_STATION_1_CYCLE".SEQUENCE.RUNNING )
      wire#w3
      S_Coil( "DB1281_UNIT_02_PART_CHECK_STATION_0".FIX_2_CLAMP_LOST_MEM )
   END_RUNG
   RUNG wire#powerrail
      Contact( "DB3600_UNIT_02_FIXTURE_2".CLAMPED_WITH_PART_ANALOG )
   END_RUNG wire#w1
   RUNG wire#w2
      I_Contact( "DB4000_FIX_TABLE_POSITIONS".UNIT_02.FIXTURE_2.IN_LOAD_UNLOAD_STATION_1 )
   END_RUNG wire#w3
   // the same network as SCL:
   #_w1 := "DB3610_U2_F2_GRIPPER".CYL.FULL_CLOSED OR "DB3600_UNIT_02_FIXTURE_2".CLAMPED_WITH_PART_ANALOG;
   #_w2 := NOT #_w1 AND "DB1281_UNIT_02_PART_CHECK_STATION_0".AUX_PULSE_3;   // falling edge
   "DB1281_UNIT_02_PART_CHECK_STATION_0".AUX_PULSE_3 := #_w1;
   IF #_w2 AND "DB8000_PART_STATUS".UNIT_02.FIXTURE_2.PART_A.STATUS.PRESENT AND NOT "DB8000_PART_STATUS".UNIT_02.FIXTURE_2.PART_A.STATUS.VIRTUAL_PART AND NOT "DB1101_MACHINE_SEQUENCE".RUNNING AND (NOT "DB1253_UNIT_02_STATION_1_CYCLE".SEQUENCE.RUNNING OR NOT "DB4000_FIX_TABLE_POSITIONS".UNIT_02.FIXTURE_2.IN_LOAD_UNLOAD_STATION_1) THEN
       "DB1281_UNIT_02_PART_CHECK_STATION_0".FIX_2_CLAMP_LOST_MEM := TRUE;
   END_IF;
END_REGION

REGION Network 10: FIXTURE 3 CLAMP LOST MEMORY
   RUNG wire#powerrail
      Contact( "DB3710_U2_F3_GRIPPER".CYL.FULL_CLOSED )
      wire#w1
      N_Trig( "DB1281_UNIT_02_PART_CHECK_STATION_0".AUX_PULSE_4 )
      Contact( "DB8000_PART_STATUS".UNIT_02.FIXTURE_3.PART_A.STATUS.PRESENT )
      I_Contact( "DB8000_PART_STATUS".UNIT_02.FIXTURE_3.PART_A.STATUS.VIRTUAL_PART )
      I_Contact( "DB1101_MACHINE_SEQUENCE".RUNNING )
      wire#w2
      I_Contact( "DB1253_UNIT_02_STATION_1_CYCLE".SEQUENCE.RUNNING )
      wire#w3
      S_Coil( "DB1281_UNIT_02_PART_CHECK_STATION_0".FIX_3_CLAMP_LOST_MEM )
   END_RUNG
   RUNG wire#powerrail
      Contact( "DB3700_UNIT_02_FIXTURE_3".CLAMPED_WITH_PART_ANALOG )
   END_RUNG wire#w1
   RUNG wire#w2
      I_Contact( "DB4000_FIX_TABLE_POSITIONS".UNIT_02.FIXTURE_3.IN_LOAD_UNLOAD_STATION_1 )
   END_RUNG wire#w3
   // the same network as SCL:
   #_w1 := "DB3710_U2_F3_GRIPPER".CYL.FULL_CLOSED OR "DB3700_UNIT_02_FIXTURE_3".CLAMPED_WITH_PART_ANALOG;
   #_w2 := NOT #_w1 AND "DB1281_UNIT_02_PART_CHECK_STATION_0".AUX_PULSE_4;   // falling edge
   "DB1281_UNIT_02_PART_CHECK_STATION_0".AUX_PULSE_4 := #_w1;
   IF #_w2 AND "DB8000_PART_STATUS".UNIT_02.FIXTURE_3.PART_A.STATUS.PRESENT AND NOT "DB8000_PART_STATUS".UNIT_02.FIXTURE_3.PART_A.STATUS.VIRTUAL_PART AND NOT "DB1101_MACHINE_SEQUENCE".RUNNING AND (NOT "DB1253_UNIT_02_STATION_1_CYCLE".SEQUENCE.RUNNING OR NOT "DB4000_FIX_TABLE_POSITIONS".UNIT_02.FIXTURE_3.IN_LOAD_UNLOAD_STATION_1) THEN
       "DB1281_UNIT_02_PART_CHECK_STATION_0".FIX_3_CLAMP_LOST_MEM := TRUE;
   END_IF;
END_REGION

REGION Network 11: FIXTURE 4 CLAMP LOST MEMORY
   RUNG wire#powerrail
      Contact( "DB3810_U2_F4_GRIPPER".CYL.FULL_CLOSED )
      wire#w1
      N_Trig( "DB1281_UNIT_02_PART_CHECK_STATION_0".AUX_PULSE_5 )
      Contact( "DB8000_PART_STATUS".UNIT_02.FIXTURE_4.PART_A.STATUS.PRESENT )
      I_Contact( "DB8000_PART_STATUS".UNIT_02.FIXTURE_4.PART_A.STATUS.VIRTUAL_PART )
      I_Contact( "DB1101_MACHINE_SEQUENCE".RUNNING )
      wire#w2
      I_Contact( "DB1253_UNIT_02_STATION_1_CYCLE".SEQUENCE.RUNNING )
      wire#w3
      S_Coil( "DB1281_UNIT_02_PART_CHECK_STATION_0".FIX_4_CLAMP_LOST_MEM )
   END_RUNG
   RUNG wire#powerrail
      Contact( "DB3800_UNIT_02_FIXTURE_4".CLAMPED_WITH_PART_ANALOG )
   END_RUNG wire#w1
   RUNG wire#w2
      I_Contact( "DB4000_FIX_TABLE_POSITIONS".UNIT_02.FIXTURE_4.IN_LOAD_UNLOAD_STATION_1 )
   END_RUNG wire#w3
   // the same network as SCL:
   #_w1 := "DB3810_U2_F4_GRIPPER".CYL.FULL_CLOSED OR "DB3800_UNIT_02_FIXTURE_4".CLAMPED_WITH_PART_ANALOG;
   #_w2 := NOT #_w1 AND "DB1281_UNIT_02_PART_CHECK_STATION_0".AUX_PULSE_5;   // falling edge
   "DB1281_UNIT_02_PART_CHECK_STATION_0".AUX_PULSE_5 := #_w1;
   IF #_w2 AND "DB8000_PART_STATUS".UNIT_02.FIXTURE_4.PART_A.STATUS.PRESENT AND NOT "DB8000_PART_STATUS".UNIT_02.FIXTURE_4.PART_A.STATUS.VIRTUAL_PART AND NOT "DB1101_MACHINE_SEQUENCE".RUNNING AND (NOT "DB1253_UNIT_02_STATION_1_CYCLE".SEQUENCE.RUNNING OR NOT "DB4000_FIX_TABLE_POSITIONS".UNIT_02.FIXTURE_4.IN_LOAD_UNLOAD_STATION_1) THEN
       "DB1281_UNIT_02_PART_CHECK_STATION_0".FIX_4_CLAMP_LOST_MEM := TRUE;
   END_IF;
END_REGION

REGION Network 12: AUTO REQUEST
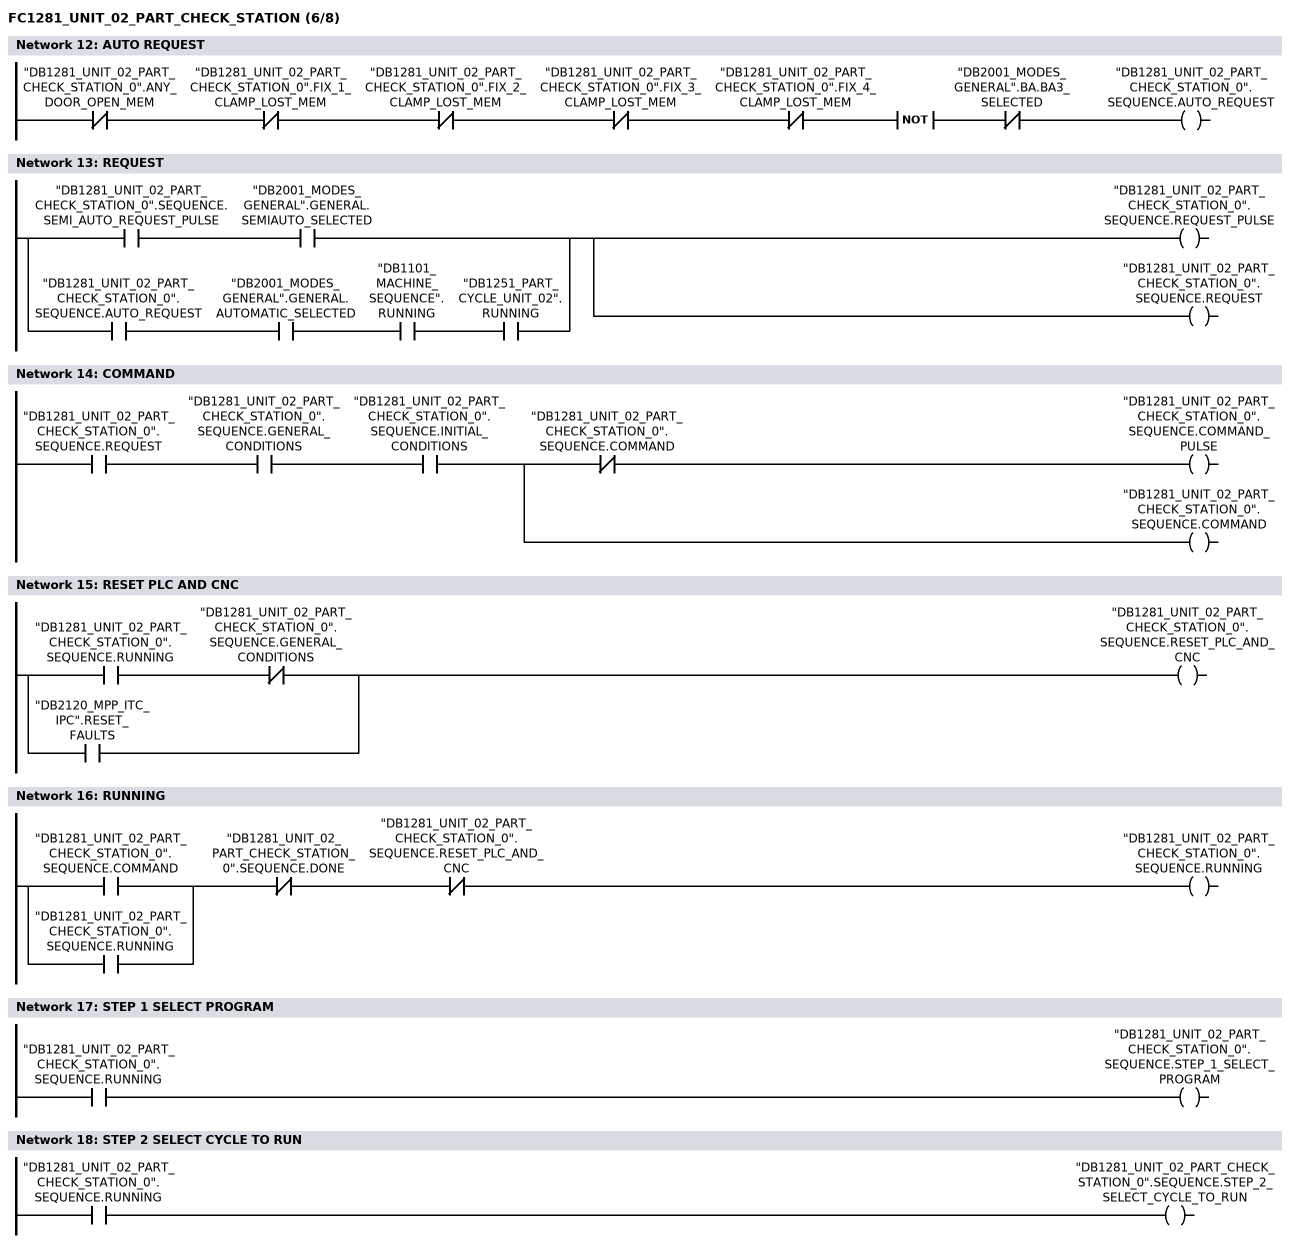
   RUNG wire#powerrail
      I_Contact( "DB1281_UNIT_02_PART_CHECK_STATION_0".ANY_DOOR_OPEN_MEM )
      I_Contact( "DB1281_UNIT_02_PART_CHECK_STATION_0".FIX_1_CLAMP_LOST_MEM )
      I_Contact( "DB1281_UNIT_02_PART_CHECK_STATION_0".FIX_2_CLAMP_LOST_MEM )
      I_Contact( "DB1281_UNIT_02_PART_CHECK_STATION_0".FIX_3_CLAMP_LOST_MEM )
      I_Contact( "DB1281_UNIT_02_PART_CHECK_STATION_0".FIX_4_CLAMP_LOST_MEM )
      Not()
      I_Contact( "DB2001_MODES_GENERAL".BA.BA3_SELECTED )
      Coil( "DB1281_UNIT_02_PART_CHECK_STATION_0".SEQUENCE.AUTO_REQUEST )
   END_RUNG
   // the same network as SCL:
   "DB1281_UNIT_02_PART_CHECK_STATION_0".SEQUENCE.AUTO_REQUEST := NOT (NOT "DB1281_UNIT_02_PART_CHECK_STATION_0".ANY_DOOR_OPEN_MEM AND NOT "DB1281_UNIT_02_PART_CHECK_STATION_0".FIX_1_CLAMP_LOST_MEM AND NOT "DB1281_UNIT_02_PART_CHECK_STATION_0".FIX_2_CLAMP_LOST_MEM AND NOT "DB1281_UNIT_02_PART_CHECK_STATION_0".FIX_3_CLAMP_LOST_MEM AND NOT "DB1281_UNIT_02_PART_CHECK_STATION_0".FIX_4_CLAMP_LOST_MEM) AND NOT "DB2001_MODES_GENERAL".BA.BA3_SELECTED;
END_REGION

REGION Network 13: REQUEST
   RUNG wire#powerrail
      Contact( "DB1281_UNIT_02_PART_CHECK_STATION_0".SEQUENCE.SEMI_AUTO_REQUEST_PULSE )
      Contact( "DB2001_MODES_GENERAL".GENERAL.SEMIAUTO_SELECTED )
      wire#w1
      Coil( "DB1281_UNIT_02_PART_CHECK_STATION_0".SEQUENCE.REQUEST_PULSE )
   END_RUNG
   RUNG wire#powerrail
      Contact( "DB1281_UNIT_02_PART_CHECK_STATION_0".SEQUENCE.AUTO_REQUEST )
      Contact( "DB2001_MODES_GENERAL".GENERAL.AUTOMATIC_SELECTED )
      Contact( "DB1101_MACHINE_SEQUENCE".RUNNING )
      Contact( "DB1251_PART_CYCLE_UNIT_02".RUNNING )
   END_RUNG wire#w1
   RUNG wire#w1
      Coil( "DB1281_UNIT_02_PART_CHECK_STATION_0".SEQUENCE.REQUEST )
   END_RUNG
   // the same network as SCL:
   "DB1281_UNIT_02_PART_CHECK_STATION_0".SEQUENCE.REQUEST_PULSE := ("DB1281_UNIT_02_PART_CHECK_STATION_0".SEQUENCE.SEMI_AUTO_REQUEST_PULSE AND "DB2001_MODES_GENERAL".GENERAL.SEMIAUTO_SELECTED) OR ("DB1281_UNIT_02_PART_CHECK_STATION_0".SEQUENCE.AUTO_REQUEST AND "DB2001_MODES_GENERAL".GENERAL.AUTOMATIC_SELECTED AND "DB1101_MACHINE_SEQUENCE".RUNNING AND "DB1251_PART_CYCLE_UNIT_02".RUNNING);
   "DB1281_UNIT_02_PART_CHECK_STATION_0".SEQUENCE.REQUEST := "DB1281_UNIT_02_PART_CHECK_STATION_0".SEQUENCE.REQUEST_PULSE;
END_REGION

REGION Network 14: COMMAND
   RUNG wire#powerrail
      Contact( "DB1281_UNIT_02_PART_CHECK_STATION_0".SEQUENCE.REQUEST )
      Contact( "DB1281_UNIT_02_PART_CHECK_STATION_0".SEQUENCE.GENERAL_CONDITIONS )
      Contact( "DB1281_UNIT_02_PART_CHECK_STATION_0".SEQUENCE.INITIAL_CONDITIONS )
      wire#w1
      I_Contact( "DB1281_UNIT_02_PART_CHECK_STATION_0".SEQUENCE.COMMAND )
      Coil( "DB1281_UNIT_02_PART_CHECK_STATION_0".SEQUENCE.COMMAND_PULSE )
   END_RUNG
   RUNG wire#w1
      Coil( "DB1281_UNIT_02_PART_CHECK_STATION_0".SEQUENCE.COMMAND )
   END_RUNG
   // the same network as SCL:
   #_w1 := "DB1281_UNIT_02_PART_CHECK_STATION_0".SEQUENCE.REQUEST AND "DB1281_UNIT_02_PART_CHECK_STATION_0".SEQUENCE.GENERAL_CONDITIONS AND "DB1281_UNIT_02_PART_CHECK_STATION_0".SEQUENCE.INITIAL_CONDITIONS;
   "DB1281_UNIT_02_PART_CHECK_STATION_0".SEQUENCE.COMMAND_PULSE := #_w1 AND NOT "DB1281_UNIT_02_PART_CHECK_STATION_0".SEQUENCE.COMMAND;
   "DB1281_UNIT_02_PART_CHECK_STATION_0".SEQUENCE.COMMAND := #_w1;
END_REGION

REGION Network 15: RESET PLC AND CNC
   RUNG wire#powerrail
      Contact( "DB1281_UNIT_02_PART_CHECK_STATION_0".SEQUENCE.RUNNING )
      I_Contact( "DB1281_UNIT_02_PART_CHECK_STATION_0".SEQUENCE.GENERAL_CONDITIONS )
      wire#w1
      Coil( "DB1281_UNIT_02_PART_CHECK_STATION_0".SEQUENCE.RESET_PLC_AND_CNC )
   END_RUNG
   RUNG wire#powerrail
      Contact( "DB2120_MPP_ITC_IPC".RESET_FAULTS )
   END_RUNG wire#w1
   // the same network as SCL:
   "DB1281_UNIT_02_PART_CHECK_STATION_0".SEQUENCE.RESET_PLC_AND_CNC := ("DB1281_UNIT_02_PART_CHECK_STATION_0".SEQUENCE.RUNNING AND NOT "DB1281_UNIT_02_PART_CHECK_STATION_0".SEQUENCE.GENERAL_CONDITIONS) OR "DB2120_MPP_ITC_IPC".RESET_FAULTS;
END_REGION

REGION Network 16: RUNNING
   RUNG wire#powerrail
      Contact( "DB1281_UNIT_02_PART_CHECK_STATION_0".SEQUENCE.COMMAND )
      wire#w1
      I_Contact( "DB1281_UNIT_02_PART_CHECK_STATION_0".SEQUENCE.DONE )
      I_Contact( "DB1281_UNIT_02_PART_CHECK_STATION_0".SEQUENCE.RESET_PLC_AND_CNC )
      Coil( "DB1281_UNIT_02_PART_CHECK_STATION_0".SEQUENCE.RUNNING )
   END_RUNG
   RUNG wire#powerrail
      Contact( "DB1281_UNIT_02_PART_CHECK_STATION_0".SEQUENCE.RUNNING )
   END_RUNG wire#w1
   // the same network as SCL:
   "DB1281_UNIT_02_PART_CHECK_STATION_0".SEQUENCE.RUNNING := ("DB1281_UNIT_02_PART_CHECK_STATION_0".SEQUENCE.COMMAND OR "DB1281_UNIT_02_PART_CHECK_STATION_0".SEQUENCE.RUNNING) AND NOT "DB1281_UNIT_02_PART_CHECK_STATION_0".SEQUENCE.DONE AND NOT "DB1281_UNIT_02_PART_CHECK_STATION_0".SEQUENCE.RESET_PLC_AND_CNC;
END_REGION

REGION Network 17: STEP 1 SELECT PROGRAM
   RUNG wire#powerrail
      Contact( "DB1281_UNIT_02_PART_CHECK_STATION_0".SEQUENCE.RUNNING )
      Coil( "DB1281_UNIT_02_PART_CHECK_STATION_0".SEQUENCE.STEP_1_SELECT_PROGRAM )
   END_RUNG
   // the same network as SCL:
   "DB1281_UNIT_02_PART_CHECK_STATION_0".SEQUENCE.STEP_1_SELECT_PROGRAM := "DB1281_UNIT_02_PART_CHECK_STATION_0".SEQUENCE.RUNNING;
END_REGION

REGION Network 18: STEP 2 SELECT CYCLE TO RUN
   RUNG wire#powerrail
      Contact( "DB1281_UNIT_02_PART_CHECK_STATION_0".SEQUENCE.RUNNING )
      Coil( "DB1281_UNIT_02_PART_CHECK_STATION_0".SEQUENCE.STEP_2_SELECT_CYCLE_TO_RUN )
   END_RUNG
   // the same network as SCL:
   "DB1281_UNIT_02_PART_CHECK_STATION_0".SEQUENCE.STEP_2_SELECT_CYCLE_TO_RUN := "DB1281_UNIT_02_PART_CHECK_STATION_0".SEQUENCE.RUNNING;
END_REGION

REGION Network 19: STEP 3 RUN CNC PROGRAM
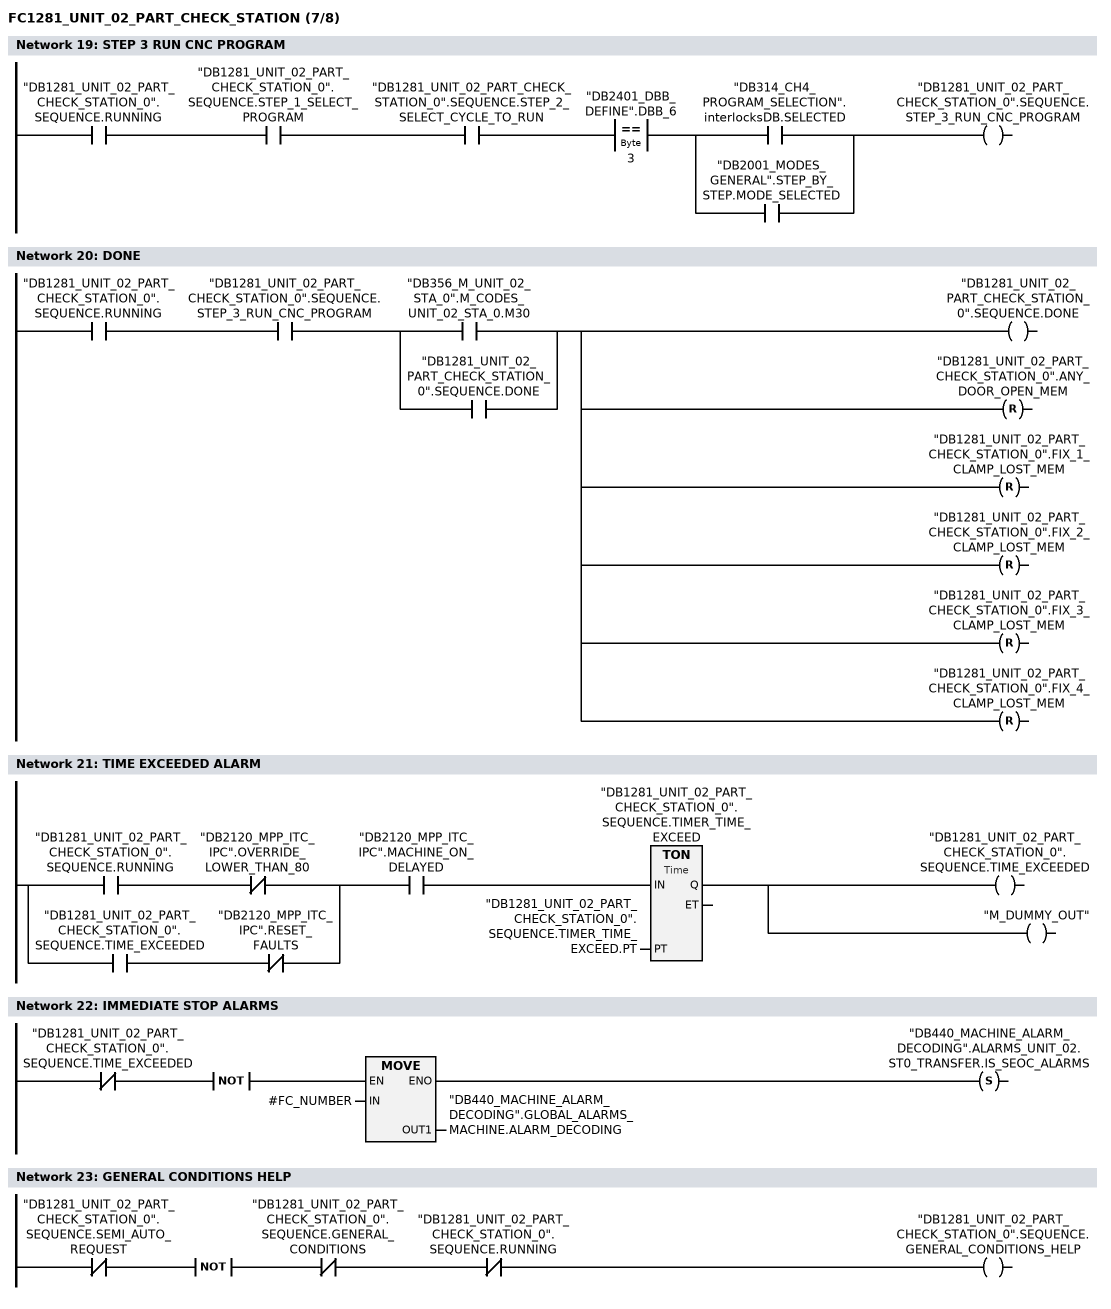
   RUNG wire#powerrail
      Contact( "DB1281_UNIT_02_PART_CHECK_STATION_0".SEQUENCE.RUNNING )
      Contact( "DB1281_UNIT_02_PART_CHECK_STATION_0".SEQUENCE.STEP_1_SELECT_PROGRAM )
      Contact( "DB1281_UNIT_02_PART_CHECK_STATION_0".SEQUENCE.STEP_2_SELECT_CYCLE_TO_RUN )
      { S7_Templates := "SrcType := Byte" } EQ_Contact(in1 := "DB2401_DBB_DEFINE".DBB_6, in2 := 3)
      wire#w1
      Contact( "DB314_CH4_PROGRAM_SELECTION".interlocksDB.SELECTED )
      wire#w2
      Coil( "DB1281_UNIT_02_PART_CHECK_STATION_0".SEQUENCE.STEP_3_RUN_CNC_PROGRAM )
   END_RUNG
   RUNG wire#w1
      Contact( "DB2001_MODES_GENERAL".STEP_BY_STEP.MODE_SELECTED )
   END_RUNG wire#w2
   // the same network as SCL:
   "DB1281_UNIT_02_PART_CHECK_STATION_0".SEQUENCE.STEP_3_RUN_CNC_PROGRAM := "DB1281_UNIT_02_PART_CHECK_STATION_0".SEQUENCE.RUNNING AND "DB1281_UNIT_02_PART_CHECK_STATION_0".SEQUENCE.STEP_1_SELECT_PROGRAM AND "DB1281_UNIT_02_PART_CHECK_STATION_0".SEQUENCE.STEP_2_SELECT_CYCLE_TO_RUN AND ("DB2401_DBB_DEFINE".DBB_6 = 3) AND ("DB314_CH4_PROGRAM_SELECTION".interlocksDB.SELECTED OR "DB2001_MODES_GENERAL".STEP_BY_STEP.MODE_SELECTED);
END_REGION

REGION Network 20: DONE
   RUNG wire#powerrail
      Contact( "DB1281_UNIT_02_PART_CHECK_STATION_0".SEQUENCE.RUNNING )
      Contact( "DB1281_UNIT_02_PART_CHECK_STATION_0".SEQUENCE.STEP_3_RUN_CNC_PROGRAM )
      wire#w1
      Contact( "DB356_M_UNIT_02_STA_0".M_CODES_UNIT_02_STA_0.M30 )
      wire#w2
      Coil( "DB1281_UNIT_02_PART_CHECK_STATION_0".SEQUENCE.DONE )
   END_RUNG
   RUNG wire#w1
      Contact( "DB1281_UNIT_02_PART_CHECK_STATION_0".SEQUENCE.DONE )
   END_RUNG wire#w2
   RUNG wire#w2
      R_Coil( "DB1281_UNIT_02_PART_CHECK_STATION_0".ANY_DOOR_OPEN_MEM )
   END_RUNG
   RUNG wire#w2
      R_Coil( "DB1281_UNIT_02_PART_CHECK_STATION_0".FIX_1_CLAMP_LOST_MEM )
   END_RUNG
   RUNG wire#w2
      R_Coil( "DB1281_UNIT_02_PART_CHECK_STATION_0".FIX_2_CLAMP_LOST_MEM )
   END_RUNG
   RUNG wire#w2
      R_Coil( "DB1281_UNIT_02_PART_CHECK_STATION_0".FIX_3_CLAMP_LOST_MEM )
   END_RUNG
   RUNG wire#w2
      R_Coil( "DB1281_UNIT_02_PART_CHECK_STATION_0".FIX_4_CLAMP_LOST_MEM )
   END_RUNG
   // the same network as SCL:
   "DB1281_UNIT_02_PART_CHECK_STATION_0".SEQUENCE.DONE := "DB1281_UNIT_02_PART_CHECK_STATION_0".SEQUENCE.RUNNING AND "DB1281_UNIT_02_PART_CHECK_STATION_0".SEQUENCE.STEP_3_RUN_CNC_PROGRAM AND ("DB356_M_UNIT_02_STA_0".M_CODES_UNIT_02_STA_0.M30 OR "DB1281_UNIT_02_PART_CHECK_STATION_0".SEQUENCE.DONE);
   IF "DB1281_UNIT_02_PART_CHECK_STATION_0".SEQUENCE.DONE THEN
       "DB1281_UNIT_02_PART_CHECK_STATION_0".ANY_DOOR_OPEN_MEM := FALSE;
       "DB1281_UNIT_02_PART_CHECK_STATION_0".FIX_1_CLAMP_LOST_MEM := FALSE;
       "DB1281_UNIT_02_PART_CHECK_STATION_0".FIX_2_CLAMP_LOST_MEM := FALSE;
       "DB1281_UNIT_02_PART_CHECK_STATION_0".FIX_3_CLAMP_LOST_MEM := FALSE;
       "DB1281_UNIT_02_PART_CHECK_STATION_0".FIX_4_CLAMP_LOST_MEM := FALSE;
   END_IF;
END_REGION

REGION Network 21: TIME EXCEEDED ALARM
   RUNG wire#powerrail
      Contact( "DB1281_UNIT_02_PART_CHECK_STATION_0".SEQUENCE.RUNNING )
      I_Contact( "DB2120_MPP_ITC_IPC".OVERRIDE_LOWER_THAN_80 )
      wire#w1
      Contact( "DB2120_MPP_ITC_IPC".MACHINE_ON_DELAYED )
      { S7_Templates := "time_type := Time" } "DB1281_UNIT_02_PART_CHECK_STATION_0".SEQUENCE.TIMER_TIME_EXCEED.TON(pt := "DB1281_UNIT_02_PART_CHECK_STATION_0".SEQUENCE.TIMER_TIME_EXCEED.PT, et =>)
      wire#w2
      Coil( "DB1281_UNIT_02_PART_CHECK_STATION_0".SEQUENCE.TIME_EXCEEDED )
   END_RUNG
   RUNG wire#powerrail
      Contact( "DB1281_UNIT_02_PART_CHECK_STATION_0".SEQUENCE.TIME_EXCEEDED )
      I_Contact( "DB2120_MPP_ITC_IPC".RESET_FAULTS )
   END_RUNG wire#w1
   RUNG wire#w2
      Coil( "M_DUMMY_OUT" )
   END_RUNG
   // the same network as SCL:
   "DB1281_UNIT_02_PART_CHECK_STATION_0".SEQUENCE.TIMER_TIME_EXCEED.TON(IN := (("DB1281_UNIT_02_PART_CHECK_STATION_0".SEQUENCE.RUNNING AND NOT "DB2120_MPP_ITC_IPC".OVERRIDE_LOWER_THAN_80) OR ("DB1281_UNIT_02_PART_CHECK_STATION_0".SEQUENCE.TIME_EXCEEDED AND NOT "DB2120_MPP_ITC_IPC".RESET_FAULTS)) AND "DB2120_MPP_ITC_IPC".MACHINE_ON_DELAYED,
                           PT := "DB1281_UNIT_02_PART_CHECK_STATION_0".SEQUENCE.TIMER_TIME_EXCEED.PT);
   "DB1281_UNIT_02_PART_CHECK_STATION_0".SEQUENCE.TIME_EXCEEDED := "DB1281_UNIT_02_PART_CHECK_STATION_0".SEQUENCE.TIMER_TIME_EXCEED.Q;
   "M_DUMMY_OUT" := "DB1281_UNIT_02_PART_CHECK_STATION_0".SEQUENCE.TIMER_TIME_EXCEED.Q;
END_REGION

REGION Network 22: IMMEDIATE STOP ALARMS
   RUNG wire#powerrail
      I_Contact( "DB1281_UNIT_02_PART_CHECK_STATION_0".SEQUENCE.TIME_EXCEEDED )
      Not()
      { S7_GenerateENO := "TRUE" } Move(in := #FC_NUMBER, out1 => "DB440_MACHINE_ALARM_DECODING".GLOBAL_ALARMS_MACHINE.ALARM_DECODING)
      S_Coil( "DB440_MACHINE_ALARM_DECODING".ALARMS_UNIT_02.ST0_TRANSFER.IS_SEOC_ALARMS )
   END_RUNG
   // the same network as SCL:
   // ENO of a box is taken as its EN; it also drops when the box reports an error
   IF NOT (NOT "DB1281_UNIT_02_PART_CHECK_STATION_0".SEQUENCE.TIME_EXCEEDED) THEN
       "DB440_MACHINE_ALARM_DECODING".GLOBAL_ALARMS_MACHINE.ALARM_DECODING := #FC_NUMBER;
       "DB440_MACHINE_ALARM_DECODING".ALARMS_UNIT_02.ST0_TRANSFER.IS_SEOC_ALARMS := TRUE;
   END_IF;
END_REGION

REGION Network 23: GENERAL CONDITIONS HELP
   RUNG wire#powerrail
      I_Contact( "DB1281_UNIT_02_PART_CHECK_STATION_0".SEQUENCE.SEMI_AUTO_REQUEST )
      Not()
      I_Contact( "DB1281_UNIT_02_PART_CHECK_STATION_0".SEQUENCE.GENERAL_CONDITIONS )
      I_Contact( "DB1281_UNIT_02_PART_CHECK_STATION_0".SEQUENCE.RUNNING )
      Coil( "DB1281_UNIT_02_PART_CHECK_STATION_0".SEQUENCE.GENERAL_CONDITIONS_HELP )
   END_RUNG
   // the same network as SCL:
   "DB1281_UNIT_02_PART_CHECK_STATION_0".SEQUENCE.GENERAL_CONDITIONS_HELP := NOT (NOT "DB1281_UNIT_02_PART_CHECK_STATION_0".SEQUENCE.SEMI_AUTO_REQUEST) AND NOT "DB1281_UNIT_02_PART_CHECK_STATION_0".SEQUENCE.GENERAL_CONDITIONS AND NOT "DB1281_UNIT_02_PART_CHECK_STATION_0".SEQUENCE.RUNNING;
END_REGION

REGION Network 24: INITIAL CONDITIONS HELP
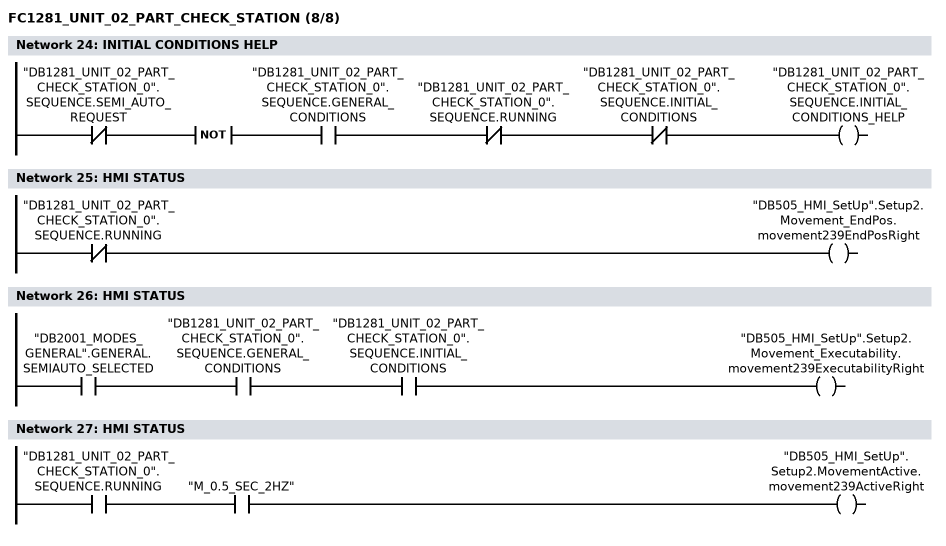
   RUNG wire#powerrail
      I_Contact( "DB1281_UNIT_02_PART_CHECK_STATION_0".SEQUENCE.SEMI_AUTO_REQUEST )
      Not()
      Contact( "DB1281_UNIT_02_PART_CHECK_STATION_0".SEQUENCE.GENERAL_CONDITIONS )
      I_Contact( "DB1281_UNIT_02_PART_CHECK_STATION_0".SEQUENCE.RUNNING )
      I_Contact( "DB1281_UNIT_02_PART_CHECK_STATION_0".SEQUENCE.INITIAL_CONDITIONS )
      Coil( "DB1281_UNIT_02_PART_CHECK_STATION_0".SEQUENCE.INITIAL_CONDITIONS_HELP )
   END_RUNG
   // the same network as SCL:
   "DB1281_UNIT_02_PART_CHECK_STATION_0".SEQUENCE.INITIAL_CONDITIONS_HELP := NOT (NOT "DB1281_UNIT_02_PART_CHECK_STATION_0".SEQUENCE.SEMI_AUTO_REQUEST) AND "DB1281_UNIT_02_PART_CHECK_STATION_0".SEQUENCE.GENERAL_CONDITIONS AND NOT "DB1281_UNIT_02_PART_CHECK_STATION_0".SEQUENCE.RUNNING AND NOT "DB1281_UNIT_02_PART_CHECK_STATION_0".SEQUENCE.INITIAL_CONDITIONS;
END_REGION

REGION Network 25: HMI STATUS
   RUNG wire#powerrail
      I_Contact( "DB1281_UNIT_02_PART_CHECK_STATION_0".SEQUENCE.RUNNING )
      Coil( "DB505_HMI_SetUp".Setup2.Movement_EndPos.movement239EndPosRight )
   END_RUNG
   // the same network as SCL:
   "DB505_HMI_SetUp".Setup2.Movement_EndPos.movement239EndPosRight := NOT "DB1281_UNIT_02_PART_CHECK_STATION_0".SEQUENCE.RUNNING;
END_REGION

REGION Network 26: HMI STATUS
   RUNG wire#powerrail
      Contact( "DB2001_MODES_GENERAL".GENERAL.SEMIAUTO_SELECTED )
      Contact( "DB1281_UNIT_02_PART_CHECK_STATION_0".SEQUENCE.GENERAL_CONDITIONS )
      Contact( "DB1281_UNIT_02_PART_CHECK_STATION_0".SEQUENCE.INITIAL_CONDITIONS )
      Coil( "DB505_HMI_SetUp".Setup2.Movement_Executability.movement239ExecutabilityRight )
   END_RUNG
   // the same network as SCL:
   "DB505_HMI_SetUp".Setup2.Movement_Executability.movement239ExecutabilityRight := "DB2001_MODES_GENERAL".GENERAL.SEMIAUTO_SELECTED AND "DB1281_UNIT_02_PART_CHECK_STATION_0".SEQUENCE.GENERAL_CONDITIONS AND "DB1281_UNIT_02_PART_CHECK_STATION_0".SEQUENCE.INITIAL_CONDITIONS;
END_REGION

REGION Network 27: HMI STATUS
   RUNG wire#powerrail
      Contact( "DB1281_UNIT_02_PART_CHECK_STATION_0".SEQUENCE.RUNNING )
      Contact( "M_0.5_SEC_2HZ" )
      Coil( "DB505_HMI_SetUp".Setup2.MovementActive.movement239ActiveRight )
   END_RUNG
   // the same network as SCL:
   "DB505_HMI_SetUp".Setup2.MovementActive.movement239ActiveRight := "DB1281_UNIT_02_PART_CHECK_STATION_0".SEQUENCE.RUNNING AND "M_0.5_SEC_2HZ";
END_REGION
END_FUNCTION
